// TwinCAT 3 PLC project MomTest
// Title: RIC_MOM
// Company: CFI
// Author: Phillip Prasinos
// ProjectVersion: 2.0.0
// Description: Mom Instance of RIC Gantry Crane
// ProgramVersion: 3.1.4020.2
// libraries:
//   Tc2_EtherCAT, * (Beckhoff Automation GmbH)
//   Tc2_MC2, * (Beckhoff Automation GmbH)
//   Tc2_SerialCom, * (Beckhoff Automation GmbH)
//   Tc2_Standard, * (Beckhoff Automation GmbH)
//   Tc2_System, * (Beckhoff Automation GmbH)
//   Tc2_SystemCX, * (Beckhoff Automation GmbH)
//   Tc2_Utilities, * (Beckhoff Automation GmbH)
//   Tc3_Interfaces, * (Beckhoff Automation GmbH)
//   Tc3_Module, * (Beckhoff Automation GmbH)
//   Tc2_System,3.4.17.0,Beckhoff Automation GmbH
// project tree:
//   DUTs/ EtherCAT_Kid.TcDUT, Patient.TcDUT
//   / FastTask.TcTTO, ParameterWriter.TcTTO
//   GVLs/ GVL_HMI.TcGVL
//   POUs/Function Blocks/ FB_CheckIn_EtherCAT.TcPOU, FB_EtherCATWriter.TcPOU, FB_HomeGantry.TcPOU, FB_Pulse.TcPOU, F_LoadDriveParameters.TcPOU, JoyStickGantryLogic.TcPOU, WirelessMove.TcPOU, P_FastTask.TcPOU
//   POUs/ HMIUpdate.TcPOU, MAIN.TcPOU, PlcTask.TcTTO, VariableValidation.TcPOU, WriteEtherCAT.TcPOU
//   POUs/Serial/ FB_SerialCom_Kiosk.TcPOU, FB_SerialCom_Remote.TcPOU, P_SerialRemote.TcPOU
// real-time tasks:
//   TASK PlcTask: cycle T#3ms, priority 2, ADS port 350
//   TASK ParameterWriter: cycle T#3ms, priority 6, ADS port 351
//   TASK FastTask: cycle T#4ms, priority 4, ADS port 352
// I/O:
//   DEVICE Device 3 (EtherCAT), AmsNetId 0.0.0.0.4.1
//     Box 1 (CX9020 EtherCAT slave) [CX9020 EtherCAT slave]
//     Box 2 (CX9020 EtherCAT slave) [CX9020 EtherCAT slave]
//     Box 3 (CX9020 EtherCAT slave) [CX9020 EtherCAT slave] (disabled)
//     Box 4 (CX9020 EtherCAT slave) [CX9020 EtherCAT slave] (disabled)
// variable links:
//   MomTest/MomTest Instance <-> Device 3 (EtherCAT)/Box 1 (CX9020 EtherCAT slave)
//     PlcTask Inputs/MAIN.JoyStickData <-> IO Inputs/Pdo Entry 11
//     PlcTask Inputs/MAIN.Kid[1].Address <-> IO Inputs/Pdo Entry 10
//     PlcTask Inputs/MAIN.Kid[1].HomedPosition_toMom <-> IO Inputs/Pdo Entry 2
//     PlcTask Inputs/MAIN.Kid[1].IsHardDownLimitReached <-> IO Inputs/Pdo Entry 5
//     PlcTask Inputs/MAIN.Kid[1].IsHardUpLimitReached <-> IO Inputs/Pdo Entry 4
//     PlcTask Inputs/MAIN.Kid[1].IsUltimateLimitReached <-> IO Inputs/Pdo Entry 3
//     PlcTask Inputs/MAIN.Kid[1].KidEstopCode <-> IO Inputs/Pdo Entry 9
//     PlcTask Inputs/MAIN.Kid[1].Load <-> IO Inputs/Pdo Entry 7
//     PlcTask Inputs/MAIN.Kid[1].MotionControllerErrorCode <-> IO Inputs/Pdo Entry 6
//     PlcTask Inputs/MAIN.Kid[1].Speed <-> IO Inputs/Pdo Entry 8
//     PlcTask Inputs/MAIN.Kid[1].UpdateWord_toMom <-> IO Inputs/Pdo Entry 1
//     PlcTask Outputs/MAIN.Kid[1].IsUltimateLimitBypassed <-> IO Outputs/Pdo Entry 6
//     PlcTask Outputs/MAIN.Kid[1].UpdateWord_FromMom <-> IO Outputs/Pdo Entry 1
//     PlcTask Outputs/MAIN.Kid[1].modeAccel_FromMom_Raw <-> IO Outputs/Pdo Entry 5
//     PlcTask Outputs/MAIN.Kid[1].modeDecel_FromMom_Raw <-> IO Outputs/Pdo Entry 7
//     PlcTask Outputs/MAIN.Kid[1].modeVel_FromMom_Raw <-> IO Outputs/Pdo Entry 4
//     PlcTask Outputs/MAIN.Kid[1].targetpos_FromMom_Raw <-> IO Outputs/Pdo Entry 2
//   MomTest/MomTest Instance <-> Device 3 (EtherCAT)/Box 2 (CX9020 EtherCAT slave)
//     PlcTask Inputs/MAIN.Kid[2].Address <-> IO Inputs/Pdo Entry 10
//     PlcTask Inputs/MAIN.Kid[2].HomedPosition_toMom <-> IO Inputs/Pdo Entry 2
//     PlcTask Inputs/MAIN.Kid[2].IsHardDownLimitReached <-> IO Inputs/Pdo Entry 5
//     PlcTask Inputs/MAIN.Kid[2].IsHardUpLimitReached <-> IO Inputs/Pdo Entry 4
//     PlcTask Inputs/MAIN.Kid[2].IsUltimateLimitReached <-> IO Inputs/Pdo Entry 3
//     PlcTask Inputs/MAIN.Kid[2].KidEstopCode <-> IO Inputs/Pdo Entry 9
//     PlcTask Inputs/MAIN.Kid[2].Load <-> IO Inputs/Pdo Entry 7
//     PlcTask Inputs/MAIN.Kid[2].MotionControllerErrorCode <-> IO Inputs/Pdo Entry 6
//     PlcTask Inputs/MAIN.Kid[2].Speed <-> IO Inputs/Pdo Entry 8
//     PlcTask Inputs/MAIN.Kid[2].UpdateWord_toMom <-> IO Inputs/Pdo Entry 1
//     PlcTask Outputs/MAIN.Kid[2].IsUltimateLimitBypassed <-> IO Outputs/Pdo Entry 6
//     PlcTask Outputs/MAIN.Kid[2].UpdateWord_FromMom <-> IO Outputs/Pdo Entry 1
//     PlcTask Outputs/MAIN.Kid[2].modeAccel_FromMom_Raw <-> IO Outputs/Pdo Entry 5
//     PlcTask Outputs/MAIN.Kid[2].modeDecel_FromMom_Raw <-> IO Outputs/Pdo Entry 7
//     PlcTask Outputs/MAIN.Kid[2].modeVel_FromMom_Raw <-> IO Outputs/Pdo Entry 4
//     PlcTask Outputs/MAIN.Kid[2].targetpos_FromMom_Raw <-> IO Outputs/Pdo Entry 2
//   MomTest/MomTest Instance <-> Device 3 (EtherCAT)/Box 3 (CX9020 EtherCAT slave)
//     PlcTask Inputs/MAIN.Kid[3].Address <-> IO Inputs/Pdo Entry 10
//     PlcTask Inputs/MAIN.Kid[3].HomedPosition_toMom <-> IO Inputs/Pdo Entry 2
//     PlcTask Inputs/MAIN.Kid[3].IsHardDownLimitReached <-> IO Inputs/Pdo Entry 5
//     PlcTask Inputs/MAIN.Kid[3].IsHardUpLimitReached <-> IO Inputs/Pdo Entry 4
//     PlcTask Inputs/MAIN.Kid[3].IsUltimateLimitReached <-> IO Inputs/Pdo Entry 3
//     PlcTask Inputs/MAIN.Kid[3].KidEstopCode <-> IO Inputs/Pdo Entry 9
//     PlcTask Inputs/MAIN.Kid[3].Load <-> IO Inputs/Pdo Entry 7
//     PlcTask Inputs/MAIN.Kid[3].MotionControllerErrorCode <-> IO Inputs/Pdo Entry 6
//     PlcTask Inputs/MAIN.Kid[3].Speed <-> IO Inputs/Pdo Entry 8
//     PlcTask Inputs/MAIN.Kid[3].UpdateWord_toMom <-> IO Inputs/Pdo Entry 1
//     PlcTask Outputs/MAIN.Kid[3].IsUltimateLimitBypassed <-> IO Outputs/Pdo Entry 6
//     PlcTask Outputs/MAIN.Kid[3].UpdateWord_FromMom <-> IO Outputs/Pdo Entry 1
//     PlcTask Outputs/MAIN.Kid[3].modeAccel_FromMom_Raw <-> IO Outputs/Pdo Entry 5
//     PlcTask Outputs/MAIN.Kid[3].modeDecel_FromMom_Raw <-> IO Outputs/Pdo Entry 7
//     PlcTask Outputs/MAIN.Kid[3].modeVel_FromMom_Raw <-> IO Outputs/Pdo Entry 4
//     PlcTask Outputs/MAIN.Kid[3].targetpos_FromMom_Raw <-> IO Outputs/Pdo Entry 2
//   MomTest/MomTest Instance <-> Device 3 (EtherCAT)/Box 4 (CX9020 EtherCAT slave)
//     PlcTask Inputs/MAIN.Kid[4].Address <-> IO Inputs/Pdo Entry 10
//     PlcTask Inputs/MAIN.Kid[4].HomedPosition_toMom <-> IO Inputs/Pdo Entry 2
//     PlcTask Inputs/MAIN.Kid[4].IsHardDownLimitReached <-> IO Inputs/Pdo Entry 5
//     PlcTask Inputs/MAIN.Kid[4].IsHardUpLimitReached <-> IO Inputs/Pdo Entry 4
//     PlcTask Inputs/MAIN.Kid[4].IsUltimateLimitReached <-> IO Inputs/Pdo Entry 3
//     PlcTask Inputs/MAIN.Kid[4].KidEstopCode <-> IO Inputs/Pdo Entry 9
//     PlcTask Inputs/MAIN.Kid[4].Load <-> IO Inputs/Pdo Entry 7
//     PlcTask Inputs/MAIN.Kid[4].MotionControllerErrorCode <-> IO Inputs/Pdo Entry 6
//     PlcTask Inputs/MAIN.Kid[4].Speed <-> IO Inputs/Pdo Entry 8
//     PlcTask Inputs/MAIN.Kid[4].UpdateWord_toMom <-> IO Inputs/Pdo Entry 1
//     PlcTask Outputs/MAIN.Kid[4].IsUltimateLimitBypassed <-> IO Outputs/Pdo Entry 6
//     PlcTask Outputs/MAIN.Kid[4].UpdateWord_FromMom <-> IO Outputs/Pdo Entry 1
//     PlcTask Outputs/MAIN.Kid[4].modeAccel_FromMom_Raw <-> IO Outputs/Pdo Entry 5
//     PlcTask Outputs/MAIN.Kid[4].modeDecel_FromMom_Raw <-> IO Outputs/Pdo Entry 7
//     PlcTask Outputs/MAIN.Kid[4].modeVel_FromMom_Raw <-> IO Outputs/Pdo Entry 4
//     PlcTask Outputs/MAIN.Kid[4].targetpos_FromMom_Raw <-> IO Outputs/Pdo Entry 2

CONFIGURATION MomTest
    RESOURCE PLC ON TwinCAT3
        TASK FastTask(INTERVAL := T#4ms, PRIORITY := 4);
        TASK ParameterWriter(INTERVAL := T#3ms, PRIORITY := 6);
        TASK PlcTask(INTERVAL := T#3ms, PRIORITY := 2);
        PROGRAM P_FastTask WITH FastTask : P_FastTask;
        PROGRAM WriteEtherCAT WITH ParameterWriter : WriteEtherCAT;
        PROGRAM MAIN WITH PlcTask : MAIN;
    END_RESOURCE
END_CONFIGURATION

// ---- DUTs/EtherCAT_Kid.TcDUT
TYPE EtherCAT_Kid :
STRUCT
	////////EtherCAT MoeAbsolute
	AxisID : INT := 0;
	//Status : FB_INIT_EtherCAT;
	//ReadStatus : FB_ReadStatus_EtherCAT := Status;
	//NcToPLC: FB_NcToPLC_Ethercat;
	
	//axisMoveAbs : FB_MoveAbsolute_EtherCAT;
	CheckIn : FB_CheckIn_EtherCAT;
	//ParameterReader : FB_EtherCATReader;
	//modeVel : DINT; //for hmi only

	// 1: System error sent from MOM
	
	//TargetPos : DINT;  //target position for move
	
	//modeAcc : DINT; //Maximum allowed Acceleration
	//modeJerk: UINT:= 80; //Maximum change in Accel per loop
	modeWindow : DINT:= 2000; //Allowed window for move to be complete
	leaveEnabled : BOOL := FALSE;
	//isBusy : BOOL := FALSE;
	//StartBit: BOOL :=FALSE;
	//RawToUU: LREAL;
//Velocity mode	profile EtherCAT Actual Values

	

	//VelDem_UU : DINT;
//Limits
	//dnUpLimit : DINT;
	//dnDownLimit: DINT;
	


	
	
	//HomeOffset_UU_R AT %I* : DINT;
	//HomeOffset_UU_W AT %Q* : DINT;
	

	CheckInt : DINT;
	bComTimeOutError : BOOL;
	//currentPosition: DINT;
	
	   RMT_EstopActivate : BOOL;
  RMT_DeadManPressed : BOOL;
  
  //EtherCAT 
    SetAdminMin : BOOL;
  SetAdminMax : BOOL;
  	  ResetCom : BOOL;
  SafteyReset : BOOL;
	UpdateWord_toMom  AT %I* : UDINT;
	HomedPosition_toMom AT %I* : DINT;
	IsUltimateLimitReached AT %I* : BYTE;
	IsHardUpLimitReached AT %I* : BYTE;
	IsHardDownLimitReached AT %I* : BYTE;
	MotionControllerErrorCode AT %I* :  UINT;


	 Load AT %I* : DINT;
	 Speed AT %I* :DINT;
	
	 KidEstopCode AT %I* : DINT;
	 		 Address AT %I*: AMSADDR;
	modeVel_FromMom : DINT;
modeAccel_FromMom : DINT;
ModeDecel_FromMom : DINT;
ScalingNumber : INT := 100; 		 
	 UpdateWord_FromMom AT %Q* : UDINT; //UpdateWord sends boolean information every cycle for quick inputs like deadman and Estop
	 targetpos_FromMom_Raw AT %Q* : DINT ; //FROM MOM
	 modeVel_FromMom_Raw AT %Q* : DINT ; //FROM MOM
	 modeAccel_FromMom_Raw AT %Q* : DINT ;
	 modeDecel_FromMom_Raw AT %Q* : DINT ;
	 IsUltimateLimitBypassed AT %Q* : BYTE;
	byPassSoftUp : BOOL;
	byPassSoftDown : BOOL;
	byPassHardup : BOOL;
	byPassHardDown : BOOL;
	byPassUltimate : BOOL;
	
	
	 //PAccel AT %I* : DINT  ;  //0x6048 vl_veloctity_acceleration
	// pDecel AT %I* : DINT ; //0x6049 vl_velocity_deceleration
	 //pVelMax AT %I* : INT; // 0x6042 vl_target_velocity
	 //OpModeCMD AT %I* : USINT := 2;; // 0x6060 Page 39 MODES OF OPERATION COMMAND 2-vl velocity mode  7 = interpolated position mode
 //pVelDem	AT %Q* : INT;
	// statusWord  AT %Q* : BITARR16; //0x6041
	// actualPos AT %Q*: DINT;// 0x6064 Position_actual_value
	// actualVel AT %Q*: DINT;
	// OpModeAct AT %Q* : USINT; // 0x6061 Page 39 MODES OF OPERATION DISPLAY read only result of changing 0x6060
	// ErrorCode AT %Q* : UINT;
	 
END_STRUCT
END_TYPE

// ---- DUTs/Patient.TcDUT
TYPE Patient :
STRUCT
	X : DINT := -10000; //patient location in mm
	Y : DINT := -10000; //patient location in mm
	ActiveSwitch: BOOL;
	AgeTimer : TON;
	AGE: TIME := T#0S;
END_STRUCT
END_TYPE

// ---- GVLs/GVL_HMI.TcGVL
{attribute 'qualified_only'}
VAR_GLOBAL PERSISTENT
	

//GantryLockWindow : DINT := 400;



//Patient{BeaconNumber}.Y
//Patient{BeaconNumber}.Active
//unJoystick1SelectNum : UINT;
//unJoystick2SelectNum : UINT;

//unJoystick1SelectNum : UINT;
//unJoystick2SelectNum : UINT;


//JoyStick1ScreenState : UINT;
//JoyStick2ScreenState : UINT;
//JoyStick1ScreenStateCommanded : INT;
//JoyStick2ScreenStateCOmmanded : INT;
//JoyStick1DeadManState : BOOL;
//JoyStick2DeadManState : BOOL;
//Joystick1ZAxisPressed : BOOL;
//JoyStick2ZAxisPressed : BOOL;
//JoyStick1SyncPressed : BOOL;
//JoyStick2SyncPressed: BOOL;
//JoyStick1Estop : BOOL;
//Joystick2Estop : BOOL;
//JoyStick1Age : TIME;
//JoyStick2Age : TIME;


//Bantry2BeaconNumber : INT;



GlobalFault_Code : INT;

GUIGlobalReset : BOOL;

	
END_VAR

VAR_GLOBAL
KioskScreenPower AT %Q* : BOOL;	
//Patient1 : Patient;
//Patient2 : Patient;
//Patient3 : Patient;
//Patient4 : Patient;
	EstopLight AT %Q* : BOOL;
Mom_Estop_Signal AT %I* : BOOL;
Kiosk_Estop_Signal AT %I* : BOOL;
END_VAR

// ---- POUs/Function Blocks/P_FastTask.TcPOU
PROGRAM P_FastTask
VAR
	
END_VAR

//MAIN.Serial1();
//MAIN.Serial2();
//MAIN.SerialRemoteFar(JoyStickNumber := GVL_HMI.unJoystick1SelectNum, Timeout := T#10S, ScreenActive => GVL_HMI.JoyStick1ScreenState);
//MAIN.SerialRemoteNear(JoyStickNumber := GVL_HMI.unJoystick2SelectNum, Timeout := T#10S, ScreenActive => GVL_HMI.JoyStick2ScreenState);

END_PROGRAM

// ---- POUs/WriteEtherCAT.TcPOU
PROGRAM WriteEtherCAT
VAR
	i : INT;
	i2 : INT;
	NetIDString : STRING;
	SymInfo  : ARRAY[1..4]  OF PLC_ReadSymInfoByName;
	SymInd : ARRAY[1..4] OF INT;
	HostFind : FB_GetHostAddrByName;
	COERead : adsread;
	Exec : BOOL;
	destaf : DINT;
END_VAR

//HostFind(sHostName := 'GANTRYKID_1', bExecute := Exec);
//FOR i := 1 TO 4 DO		
//	NetIDString :=INT_TO_STRING(BYTE_TO_INT(main.Kid[i].Address.netId[0]));
//
//	FOR i2 := 1 TO 5 DO NetIDString := CONCAT(Concat(netIDString, '.'), INT_TO_STRING(BYTE_TO_INT(main.Kid[i].Address.netId[i2]))); END_FOR
//SymInfo[i](NetID := NetIDString,  PORT:= main.kid[i].address.port, SymName:= 'TIID^Device 3 (EtherCAT Slave)^Outputs^CurrentPosition_ToMom', Start:=Exec);

	//MAIN.Kid[i].EtherCATWriter();
//END_FOR 	
//COERead(netid:=NetIDString, Port:=851, IDxGRP:=50593872,idxoffs:= 2164260877,Len:=4,DestAddr:=ADR(destaf),read:=Exec);

END_PROGRAM

// ---- POUs/MAIN.TcPOU
 PROGRAM MAIN
VAR_INPUT PERSISTENT
	Kid : ARRAY [1..6] OF EtherCAT_Kid;

END_VAR

VAR_INPUT
	JoyStickData AT %I* : DINT;
	JoyStickReading : DINT;
	ck : int;
	tcRestart : PLC_Reset;
		NumKids : INT := 2;
	GlobalEstopActive : BOOL;
	GlobalEstopCode : INT;
	GlobalEstopReason : STRING(255);
	JoyStickEstopActive : BOOL;
	StartHome1 : BOOL;
	Homing_Active : BOOL;
	StartHome2 : BOOL;
		xtar : DINT;
	ytar : DINT;
		JoyStick1DeadMan : BOOL;
	JoyStick2DeadMan : BOOL;
	jsResetter : BOOL;
	onUpLimit : BOOL;
	onDownLimit : BOOL;
END_VAR
VAR
	maxError : INT;
	ProcStart : NT_StartProcess;
	fbUpsPulse: FB_Pulse;

		MaxTimeOut_Reset : BOOL;
	fbWritePersistentData: FB_WritePersistentData;
		
	GantryCollision : BOOL;

	Mom_Estop_State : BOOL;
	//GantryClearanceWindow : DINT := 450;
	//HomeGantry : FB_HomeGantry;
	//HomeCarriage : FB_HomeGantry;
	TimeOutCheck : TIME;
	MaxTimeOut : Time;
	//	Kid : ARRAY [1..4] OF EtherCAT_Kid;
	//DeadMan : BOOL;
	//EStop : BOOL;
	//MAIN. : STRING(5000);
	
	i: DINT;
	Initialized : BOOL := FALSE;
	Serial1 : FB_SerialCom_Remote;
	Serial2 : FB_SerialCom_Kiosk;
	//Patient1 : Patient;
	//Patient2 : Patient;
	//Patient3 : Patient;
	//Patient4 : Patient;
	

	InterOpTimer : TON;
	TimeOutSwitch : BOOL;
	InterOpTimeout : BOOL;
	Execute : BOOL := true;
	GlobalReset : BOOL;
	ResetCount : INT;



	IN: INT;

	//HMIUpdate : HMIUpdate;
	//SerialRemoteFar : FB_SerialCom_Remote;
	//SerialRemoteNear : FB_SerialCom_Remote;
	
	//JS1 : JoyStickGantryLogic;
	//JS2 : JoystickGantryLogic;
	checker : DINT;
END_VAR



IF main.JoyStickEstopActive THEN main.GlobalEstopActive := TRUE;END_IF
IF NOT Initialized THEN
	//ProcStart(PathStr:='C:\users\administrator\desktop\setup.exe', dirname := 'C:\users\administrator\desktop', Start := TRUE);
	FOR i := 1 TO NumKids DO		
		MAIN.Kid[i].Checkin.KidID := DINT_TO_INT(i);	
		MAIN.Kid[i].AxisID := DINT_TO_INT(i); 
		KID[I].targetpos_FromMom_Raw := KID[I].HomedPosition_toMom;
		KID[i].leaveEnabled := FALSE;
	END_FOR 	
	Initialized := TRUE;
	RETURN;
END_IF


//HMIUpdate();

InterOpTimer(IN:= TimeOutSwitch, PT:= T#1000S, Q=> InterOpTimeout, ET=> TimeOutCheck);

if MaxTimeOut_Reset then MaxTimeOut := T#0s; MaxTimeOut_Reset := FALSE; END_IF
IF TimeOutCheck > MaxTimeOut THEN MaxTimeout := TimeOutCheck; END_IF

IF NOT TimeOutSwitch THEN TimeOutSwitch := NOT InterOpTimeout OR NOT TimeOutSwitch; END_IF
IF InterOpTimeOut THEN GlobalEstopActive := TRUE; GlobalEstopReason := 'INTEROPTIMEOUT'; END_IF


Joystick1Deadman := Joystick1Deadman AND NOT InterOpTimeout;




FOR i := 1 TO NumKids DO
	//MAIN.Kid[i].targetpos_FromMom_Raw := MAIN.Kid[1].HomedPosition_toMom;

	IF JoyStickData > 98304 AND JoyStickData <> 10000 THEN 
		
		MAIN.Kid[i].RMT_DeadManPressed := TRUE; 
	ELSIF JoyStickData <> 10000 THEN
		MAIN.Kid[i].RMT_DeadManPressed := FALSE;
	END_IF
	
	IF JoyStickData > 98304 THEN 
			
			JoyStickReading := (JoyStickData -98304 - 10000);
			MAIN.Kid[1].modeVel_FromMom_Raw := ABS((JoyStickReading * 1500)/10000);
			MAIN.Kid[1].modeAccel_FromMom_Raw := 3 * (((ABS(JoyStickReading) * 1200)/10000) +20);
			MAIN.Kid[1].modeDecel_FromMom_Raw := 3 * 1200;
			MAIN.Kid[1].targetpos_FromMom_Raw := MAIN.Kid[1].HomedPosition_toMom + JoyStickReading/20;	
	END_IF
		
	IF MAIN.Kid[i].modeAccel_FromMom_Raw < 10 THEN Kid[i].modeAccel_FromMom_Raw := 10; END_IF 
	//IF globalestopactive THEN kid[i].targetpos_FromMom_Raw := kid[i].HomedPosition_toMom; END_IF
	IF GVL_HMI.GUIGlobalReset THEN GlobalReset := TRUE; GVL_HMI.GUIGlobalReset := FALSE; END_IF
	IF GlobalReset THEN
		MAIN.Kid[i].resetCOM := TRUE;
		MAIN.Kid[i].SafteyReset := TRUE;
		MAIN.Kid[i].bComTimeOutError := FALSE;
		Kid[i].RMT_EstopActivate :=Mom_Estop_State;
		InterOpTimeOut := FALSE;
		timeoutSwitch := FALSE;
		GlobalEstopActive := false;
		GlobalEstopCode := 0;
		joystickEstopActive := False;
	END_IF
	
	IF Execute THEN
		MAIN.Kid[i].CheckIn.momControl := TRUE;
		IF(TimeOutCheck > T#500MS ) THEN   //this is the maximum allowed timeout when a deadman is pressed
			MAIN.Kid[i].RMT_DeadManPressed := FALSE;
		END_IF
	ELSE
		MAIN.Kid[i].CheckIn.momControl := FALSE;
		MAIN.Kid[i].RMT_DeadManPressed := FALSE;
	END_IF
	
		MAIN.Kid[i].CheckIn();
END_FOR 

IF GlobalReset AND NOT 
((Kid[1].CheckIn.momControl_FromKid AND(MAIN.Kid[1].Checkin.SafteyTripped  OR kid[1].checkin.CommError_FromKid)) OR 
 (Kid[2].CheckIn.momControl_FromKid AND (Kid[2].Checkin.SafteyTripped OR kid[2].checkin.CommError_FromKid)) OR
//(Kid[3].CheckIn.momControl_FromKid AND(Kid[3].Checkin.SafteyTripped OR kid[3].checkin.CommError_FromKid)) OR
//(Kid[4].CheckIn.momControl_FromKid AND(Kid[4].Checkin.SafteyTripped OR kid[4].checkin.CommError_FromKid)) OR
//(Kid[5].CheckIn.momControl_FromKid AND(Kid[5].Checkin.SafteyTripped OR kid[5].checkin.CommError_FromKid)) OR
//(Kid[6].CheckIn.momControl_FromKid AND(Kid[6].Checkin.SafteyTripped OR kid[6].checkin.CommError_FromKid)) OR
						GlobalEstopActive)  THEN
	GlobalReset:= FALSE;
	ResetCount := 0;
ELSIF GlobalReset THEN
	GlobalEstopActive := FALSE;
	ResetCount := ResetCount + 1;
	IF ResetCount > 300 THEN GlobalReset := FALSE; ResetCount := 0; END_IF
END_IF



//JS1(HookX := kid[1], HookY := Kid[2], sm := SerialRemoteFar); js1.Patient[1] := GVL_HMI.Patient1; js1.Patient[2] := GVL_HMI.Patient2; js1.Patient[3] := GVL_HMI.Patient3; js1.Patient[4] := GVL_HMI.Patient4;
//JS2(HookX := kid[3], HookY := Kid[4], sm := SerialRemoteNear); js2.Patient[1] := GVL_HMI.Patient1; js2.Patient[2] := GVL_HMI.Patient2; js2.Patient[3] := GVL_HMI.Patient3; js2.Patient[4] := GVL_HMI.Patient4;

checker := checker + 1;

i :=  Kid[1].HomedPosition_toMom; i := Kid[1].targetpos_FromMom_Raw; i := Kid[1].ScalingNumber; i := Kid[1].modeAccel_FromMom_RAW; i := Kid[1].modeVel_FromMom_RAW; i := Kid[1].ModeDecel_FromMom_RAW;
i :=  Kid[2].HomedPosition_toMom;  i := Kid[2].targetpos_FromMom_Raw;i := Kid[2].ScalingNumber; i := Kid[2].modeAccel_FromMom_RAW; i := Kid[2].modeVel_FromMom_RAW; i := Kid[2].ModeDecel_FromMom_RAW;
i :=  Kid[3].HomedPosition_toMom;  i := Kid[3].targetpos_FromMom_Raw;i := Kid[3].ScalingNumber; i := Kid[3].modeAccel_FromMom_RAW; i := Kid[2].modeVel_FromMom_RAW; i := Kid[3].ModeDecel_FromMom_RAW;
i :=  Kid[4].HomedPosition_toMom; i := Kid[4].targetpos_FromMom_Raw;  i := Kid[4].ScalingNumber; i := Kid[4].modeAccel_FromMom_RAW; i := Kid[2].modeVel_FromMom_RAW; i := Kid[3].ModeDecel_FromMom_RAW;




i := MAIN.Kid[1].UpdateWord_toMom;
i := MAIN.Kid[2].UpdateWord_toMom;
i := MAIN.Kid[3].UpdateWord_toMom;
i := MAIN.Kid[4].UpdateWord_toMom;
i := MAIN.Kid[5].UpdateWord_toMom;
i := MAIN.Kid[6].UpdateWord_toMom;


WriteEtherCAT();

fbUpsPulse(bEnable:= TRUE, tTimeOn:= T#100MS, tTimeOff:= T#30S, bPulse=> );


	in := in + 1;
	
	i := 2;
	ck :=DINT_TO_INT(Kid[1].targetpos_FromMom_Raw );
IF MAIN.Kid[1].targetpos_FromMom_Raw < 0 THEN  MAIN.Kid[1].targetpos_FromMom_Raw := 0; END_IF
IF MAIN.Kid[1].targetpos_FromMom_Raw > 12000 THEN  MAIN.Kid[1].targetpos_FromMom_Raw := 0; END_IF

	FOR i := 1 TO NumKids DO
		
		IF ABS(MAIN.Kid[i].HomedPosition_toMom - MAIN.Kid[1].HomedPosition_toMom) > maxError THEN maxError := DINT_TO_INT(ABS(MAIN.Kid[i].HomedPosition_toMom - MAIN.Kid[1].HomedPosition_toMom)); END_IF
		MAIN.Kid[i].targetpos_FromMom_Raw := MAIN.Kid[1].targetpos_FromMom_Raw;
		MAIN.Kid[i].modeVel_FromMom_Raw := MAIN.Kid[1].modeVel_FromMom_Raw + (ABS((MAIN.Kid[i].HomedPosition_toMom - MAIN.Kid[1].HomedPosition_toMom)) MOD 100);
		MAIN.Kid[i].modeAccel_FromMom_Raw := MAIN.Kid[1].modeAccel_FromMom_Raw + ABS((MAIN.Kid[i].HomedPosition_toMom - MAIN.Kid[1].HomedPosition_toMom)) MOD 50;
		MAIN.Kid[i].modeDecel_FromMom_Raw := MAIN.Kid[1].modeDecel_FromMom_Raw + ABS((MAIN.Kid[i].HomedPosition_toMom - MAIN.Kid[1].HomedPosition_toMom)) MOD 50;
		MAIN.Kid[i].ScalingNumber := MAIN.Kid[1].ScalingNumber;
		MAIN.Kid[i].RMT_DeadManPressed := MAIN.Kid[1].RMT_DeadManPressed;
		onDownLimit := FALSE;
		onUpLimit := FALSE;
		IF(MAIN.Kid[i].IsHardDownLimitReached> 0 AND MAIN.Kid[i].targetpos_FromMom_Raw <= MAIN.Kid[1].targetpos_FromMom_Raw) THEN onDownLimit := TRUE; END_IF
		IF(MAIN.Kid[i].IsHardUpLimitReached > 0 AND MAIN.Kid[i].targetpos_FromMom_Raw >= MAIN.Kid[1].targetpos_FromMom_Raw) THEN onUpLimit := TRUE; END_IF
	END_FOR
	
	
	FOR i := 1 TO NumKids DO
		IF(onUpLimit OR onDownLimit) THEN 
		   MAIN.Kid[i].RMT_DeadManPressed := FALSE;
 // MAIN.GlobalEstopActive := TRUE;
		END_IF
	END_FOR
	
	IF JoyStickData = 10000 AND NOT jsResetter  THEN jsResetter :=TRUE; GlobalEstopActive := TRUE; jsResetter := TRUE; END_IF
	IF jsResetter AND JoyStickData <> 10000 THEN GlobalReset := TRUE; jsResetter := FALSE; END_IF
	//IF TimeOutCheck > T#60S THEN
	//	tcRestart(RESET := TRUE);
	//END_IF

END_PROGRAM

// ---- POUs/Function Blocks/FB_Pulse.TcPOU
FUNCTION_BLOCK FB_Pulse
VAR_INPUT
	bEnable		: BOOL;		//When TRUE, bPulse will be on for tTimeOn and off for tTimeOff
	tTimeOn		: TIME;		//Time bPulse is On
	tTimeOff	: TIME;		//Time bPulse is Off
END_VAR
VAR_OUTPUT
	bPulse		: BOOL;
END_VAR
VAR
	fbTON		: TON;
	fbTOF		: TOF;
END_VAR

(*
//*****************************************************************Notes**********************************************************\\



  
  
//*****************************************************************Revs**********************************************************\\
   (          who            )(    Date    ) (   Rev     ) (								Disc						)
     Chris Mauban			 	2016.05.06		0.00.01		Initial Code
				
     		 								 				
	 						
	
//*****************************************************************Code**********************************************************\\
*)
fbTON(IN:= bEnable AND NOT fbTOF.Q, PT:= tTimeOn, Q=> , ET=> );
fbTOF(IN:= fbTON.Q, PT:= tTimeOff, Q=> , ET=> );

IF bEnable THEN
	bPulse := fbTON.M;
ELSE
	bPulse := FALSE;
END_IF

END_FUNCTION_BLOCK

// ---- POUs/Serial/FB_SerialCom_Remote.TcPOU
FUNCTION_BLOCK FB_SerialCom_Remote

VAR
	x : INT :=0; 
	FRAME : ARRAY [1..10 ] OF BYTE ; 
	TxBuffer	: ComBuffer;
	RxBuffer	: ComBuffer;
		NextOffset : INT;
	yRead : INT;
	xRead : INT; 
	ButtonStateRead : INT;
	ScreenStateRead : INT;
	bCount: INT;
		(* background communication with the EL6001 terminal *)
	fbEL6002Ctrl		: SerialLineControl;
	(* 	I/O variables for a EL6001 terminal*)
	stIn_EL6002B AT %I*	: EL6inData22B;	(* linked to the EL6001 in the TwinCAT System Manager *)
	stOut_EL6002B AT %Q*	: EL6outData22B;(* linked to the EL6001 in the TwinCAT System Manager *)
	SendTimer		: TON;
	fbSend		: SendString;
	bSendBusy	: BOOL;
	eSendErrorID: ComError_t;
	fbReceive		: ReceiveData;
	AgeTimer : TON;
	Disconnected : BOOL;
	CalmDown : TIME := T#900MS;
END_VAR

VAR_INPUT
	Timeout : TIME := T#3S; //Timespan to concider the remote disconnected
	sSendString: STRING;
	ScreenCommanded : BYTE;
	JoyStickNumber : INT;
END_VAR

VAR_OUTPUT
	yAxis : INT:=0; //Up/Down result of Joystick 50 to -50
	xAxis : INT:=0; //Left/Right Result of Joystick 50 to -50
	DeadmanPressed: INT:=0; //Resulting consecutive frames with DeadmanPressed (Positive) or not pressed 
	EstopPressed: INT:=0; //Resulting consecutive frames with DeadmanPressed (Positive) or not pressed 
	ZAxisPressed: INT:=0; //Resulting consecutive frames with DeadmanPressed (Positive) or not pressed 
	SyncPressed : INT:=0; //Resulting consecutive frames with DeadmanPressed (Positive) or not pressed 
	Age : TIME;
	Connected : BOOL;
	ScreenActive : INT;
END_VAR


(* background communication with the EL6001 terminal *)
AgeTimer(IN:=TRUE, PT := Timeout, ET=> AGE, Q=> Disconnected); Connected := NOT Disconnected;

fbEL6002Ctrl(	Mode:= SERIALLINEMODE_EL6_22B, 	pComIn:= ADR(stIn_EL6002B),	pComOut:= ADR(stOut_EL6002B), 	SizeComIn:= SIZEOF(stIn_EL6002B), 	TxBuffer:= TxBuffer, 	RxBuffer:= RxBuffer, );

// Call the send block every second to repeat the transmission.
// Also call the block as long as it is busy to finish a transmission.
IF ScreenActive = ScreenCommanded OR LEN(sSendString)> 2 OR txbuffer.count > 5 THEN
	SendTimer(IN:=TRUE, PT := T#50MS + CalmDown);
	
	ELSE
	SendTimer(IN:=TRUE, PT := T#50MS );

END_IF
IF TXBuffer.Count > 10 THEN sSendString := ''; END_IF
IF SendTimer.Q OR bSendBusy THEN
	SendTimer(IN:=FALSE); (* reset timer *)
	fbSend(	SendString:=  sSendString,	TXbuffer:= TxBuffer,	Busy=> bSendBusy,	Error=> );
	IF fbSend.Error <> COMERROR_NOERROR THEN
		eSendErrorID := fbSend.Error;
	END_IF
END_IF


IF RxBuffer.Count > 9 THEN
	//IF LEN(sSendString) <= 1 THEN sSendString := ''; END_IF
	fbReceive(pReceiveData :=ADR(FRAME), SizeReceiveData := SIZEOF(FRAME),	 DataReceived =>,	 RxBuffer := RXBUFFER);
	FOR X := 1 TO 5 DO
		IF FRAME[x]= 116 AND FRAME[x+1] = 100 AND FRAME[x + 2]= 114 AND FRAME[x+3]=58  THEN sSendString := CONCAT(DINT_TO_STRING(100000 + JoyStickNumber), '$R$N');  END_IF //filter:
		IF FRAME[x]= 76 AND FRAME[x+1] = 79 AND FRAME[x + 2]= 83 AND FRAME[x+3]=83 THEN sSendString := CONCAT(DINT_TO_STRING(100000 + JoyStickNumber), '$R$N');  END_IF  //RF LOSS
		IF FRAME[x] = 10 AND FRAME[x+5] = 13 THEN
			//IF ScreenCommanded = 74 THEN sSendString := 'J' ; END_IF
sSendString := F_ToChR(ScreenCommanded); 
			
			yRead := FRAME[x+1] ;
			xRead := FRAME[x+2];
			ButtonStateRead := BYTE_TO_INT(Frame[x+3]);
			ScreenStateRead := Frame[x+4];
			
		//IF ((ButtonStateRead + xAxis + yAxis + ScreenStateRead) MOD 2)  = BOOL_TO_INT(ButtonStateRead > 64) THEN 
				ButtonStateRead := ButtonStateRead MOD 64;   //buttonstates 7th bit is used for parity 0==odd 1==even (64 = EVEN) 
				yAxis := yRead -150;
				xAxis := xRead - 150;
				NextOffSet := X;
				ScreenActive := ScreenStateRead;
				IF ButtonStateRead >= 32 THEN SyncPressed := BOOL_TO_INT(SyncPressed <=0) * (SyncPressed -1); ButtonStateRead := ButtonStateRead - 32; ELSE SyncPressed := BOOL_TO_INT(SyncPressed >=0) * (SyncPressed + 1); END_IF
				IF ButtonStateRead >= 16  THEN ZAxisPressed := BOOL_TO_INT(ZAxisPressed <=0) * (ZAxisPressed -1); ButtonStateRead := ButtonStateRead - 16; ELSE ZAxisPressed := BOOL_TO_INT(ZAxisPressed >=0) *(ZaxisPressed + 1); END_IF
				IF ButtonStateRead < 8  THEN EstopPressed := BOOL_TO_INT(EstopPressed<= 0) * (EstopPressed -1);  ELSE EStopPressed := BOOL_TO_INT(EStopPressed >= 0) * (EStopPressed + 1); ButtonStateRead := (ButtonStateRead - 8); END_IF
				IF ButtonStateRead >= 3  THEN DeadManPressed :=  BOOL_TO_INT(DeadManPressed <= 0) *(DeadManPressed - 1); ButtonStateRead := ButtonStateRead - 4; ELSE DeadmanPressed := BOOL_TO_INT(DeadManPressed >= 0) * (DeadmanPressed + 1); END_IF
				IF SyncPressed > 100 THEN SyncPressed := 100; END_IF; IF SyncPressed < -100 THEN SyncPressed := -100; END_IF
				IF ZAxisPressed > 1000 THEN ZAxisPressed := 100; END_IF; IF ZAxisPressed < -1000 THEN ZAxisPressed := -100; END_IF
				IF EStopPressed > 1000 THEN EStopPressed := 100; END_IF; IF EStopPressed < -1000 THEN EStopPressed := -100; END_IF
				IF DeadManPressed > 1000 THEN DeadManPressed := 100; END_IF; IF DeadManPressed < -1000 THEN DeadManPressed := -100; END_IF
				AgeTimer(in:=False);
			//FRAME[X+ 1] :=0; FRAME[X+ 2] :=0; FRAME[X+ 3] :=0; FRAME[X+ 4] :=0; FRAME[X+ 5] :=0;
		//	ELSE 
					bCount := bCount +1;
					
					
			//END_IF
			
			
		END_IF
		FRAME[X] :=0;
	END_FOR

END_IF

IF AgeTimer.Q THEN 
	ScreenActive := 72;
	//ScreenCommanded := 72; 
	sSendString := CONCAT(DINT_TO_STRING(100000 + JoyStickNumber), '$R$N');
ELSIF sCREENcOMMANDED = 72 THEN
	//ScreenCommanded := 73;
 END_IF
//	Age := Age + T#1MS; //IF THIS IS NOT THE CYCLE TIME OF THE TASK IT WILL NOT BE ACCURATE;

IF ScreenActive = 0 THEN ScreenActive := 72; END_IF

END_FUNCTION_BLOCK

// ---- POUs/Serial/FB_SerialCom_Kiosk.TcPOU
FUNCTION_BLOCK FB_SerialCom_Kiosk

VAR
	begpack : bool;
	x : INT;
	prefix : STRING := '$R$N';
	suffix : STRING := '$R$N';
	fcount : DINT :=0;
	FRAME : ARRAY [1..200 ] OF BYTE ; 
	swCheck0 : STRING;
	swCheck1 : STRING;
	swCheck2 : STRING;
	swCheck3 : STRING;
	swCheck4 : STRING;
	swCheck5 : STRING;
	ReceiveByte : ReceiveByte;
	LastReceivedByte : BYTE;
	TxBuffer	: ComBuffer;
	RxBuffer	: ComBuffer;

		(* background communication with the EL6001 terminal *)

		fbEL6002Ctrl		: SerialLineControl;
	bEL6002CtrlError	: BOOL;
	eEL6002CtrlErrorID	: ComError_t;
	(* 	I/O variables for a EL6001 terminal*)
	stIn_EL6002 AT %I*	: EL6inData22B;	(* linked to the EL6001 in the TwinCAT System Manager *)
	stOut_EL6002 AT %Q*	: EL6outData22B;(* linked to the EL6001 in the TwinCAT System Manager *)
	stIn_EL6002B AT %I*	: EL6inData22B;	(* linked to the EL6001 in the TwinCAT System Manager *)
	stOut_EL6002B AT %Q*	: EL6outData22B;(* linked to the EL6001 in the TwinCAT System Manager *)
	Timer		: TON;
	fbSend		: SendString;
	bSendBusy	: BOOL;
	eSendErrorID: ComError_t;

	fbReceive		: ReceiveData;
fbReceivestr		: ReceiveSTRING;


	eReceiveErrorID	: ComError_t;
	nReceiveCounter	: UDINT;

	fbF_Trig: F_TRIG;
	nStringLength: INT;
	sStringWithoutPrefix: STRING(255);

END_VAR

VAR_INPUT
	bEnable : BOOL;
	sSendString: STRING;
END_VAR

VAR_OUTPUT
	bStringReceived	: BOOL;
	sReceivedString	: STRING;
	sLastReceivedString: STRING := 'NULL';
	bDone : BOOL;
END_VAR

(*
The SerialLineControl function block is supposed to be called in every PLC cycle.
It communicates with the serial line hardware device and transmits or receives data.
The SerialLineControl can be called in the standard task (e.g.for PcCOM port usage) 
or in a separate fast task (e.g.for terminal usage) as well.
A fast separate task will be necessary at high baud rates or with KL6001 terminals 
which have a small process image (3 or 5 data bytes only)
*)

(* background communication with the EL6001 terminal *)

fbEL6002Ctrl(
	Mode:= SERIALLINEMODE_EL6_22B, 
	pComIn:= ADR(stIn_EL6002), 
	pComOut:= ADR(stOut_EL6002), 
	SizeComIn:= SIZEOF(stIn_EL6002), 
	Error=> , 
	ErrorID=> , 
	TxBuffer:= TxBuffer, 
	RxBuffer:= RxBuffer, );
IF fbEL6002Ctrl.Error THEN
	bEL6002CtrlError := TRUE;
	eEL6002CtrlErrorID := fbEL6002Ctrl.ErrorID;
END_IF


// Call the send block every second to repeat the transmission.
// Also call the block as long as it is busy to finish a transmission.
Timer(IN:=bEnable, PT := T#125MS);
IF Timer.Q OR bSendBusy THEN
	Timer(IN:=FALSE); (* reset timer *)
	fbSend(	SendString:= sSendString,
			TXbuffer:= TxBuffer,
			Busy=> bSendBusy,
			Error=> );
	IF fbSend.Error <> COMERROR_NOERROR THEN
		eSendErrorID := fbSend.Error;
	END_IF
END_IF

fbF_Trig(CLK:=bSendBusy);
bDone := bSendBusy;
	
//	Receive string data:
//	The block receives any data strings beginning with a STX ($02) and ending with an ETX ($03) character.	
//fbEL6002Ctrl.RxBuffer.Count

WHILE RxBuffer.Count > 205 AND ReceiveByte.ReceivedByte <> 150  DO			
	ReceiveByte( RxBuffer := RXBuffer);
END_WHILE

IF RxBuffer.Count > 199 THEN
fbReceive(//pPrefix := ADR(prefix),
		  //psuffix := ADR(SUFFIX),
		 //LenPrefix := 2,
		 pReceiveData :=ADR(FRAME),
		 SizeReceiveData := SIZEOF(FRAME),
		 DataReceived =>,
		 RxBuffer := RXBUFFER);
		 END_IF
		 
	IF (Frame[1] = 78 OR frame[2] = 78 OR frame[3] = 78) AND NOT GVL_HMI.KioskScreenPower  THEN
		GVL_HMI.KioskScreenPower := TRUE;
	ELSIF (Frame[1] = 70 OR frame[2] = 70 OR frame[3] = 70) AND  GVL_HMI.KioskScreenPower  THEN
			GVL_HMI.KioskScreenPower := FALSE;

	END_IF



(*
fbReceivestr(
	Prefix:= '$N',//'$02',
	Suffix:= '$R',//'$03',
	Timeout:= T#1s,
	ReceivedString:= sReceivedString,
	RXbuffer:= RxBuffer,
	StringReceived=> bStringReceived,
	Busy=> bReceiveBusy,
	Error=> ,
	RxTimeout=> bReceiveTimeout );





	//ReceiveByte(RxBuffer := RXBuffer);
	
		begPack := FALSE;
	 //CLEAR OUT BUFFER TO PREVENT OVERRUN
		ReceiveByte( RxBuffer := RXBuffer);
		IF ReceiveByte.ReceivedByte = 13 THEN
			swCheck2 := BYTE_TO_STRING(ReceiveByte.ReceivedByte);
			WHILE RxBuffer.Count > 5 AND begpack = FALSE DO //CLEAR OUT BUFFER TO PREVENT OVERRUN
				
					begPack := TRUE;
					fcount := fcount + 1;
					
					ELSE
					
							swCheck1 := BYTE_TO_STRING(ReceiveByte.ReceivedByte);
					fcount := fcount - 1;
				END_IF
			END_WHILE
			ELSE
				swCheck3 := BYTE_TO_STRING(ReceiveByte.ReceivedByte);

		END_IF
	END_WHILE
	

	
	IF begPack AND RxBuffer.Count > 4 THEN
		
				ReceiveByte( RxBuffer := RXBuffer);
				//swCheck2 := BYTE_TO_STRING(ReceiveByte.ReceivedByte);
				IF ReceiveByte.ByteReceived  AND ReceiveByte.ReceivedByte > 50 THEN yRead := BYTE_TO_INT(ReceiveByte.ReceivedByte) ; END_IF
				ReceiveByte(RxBuffer := RXBuffer);
				//swCheck3 := BYTE_TO_STRING(ReceiveByte.ReceivedByte);
				IF ReceiveByte.ByteReceived  AND ReceiveByte.ReceivedByte >50 THEN xRead := BYTE_TO_INT(ReceiveByte.ReceivedByte) ; END_IF
				ReceiveByte( RxBuffer := RXBuffer);
				//swCheck4 := BYTE_TO_STRING(ReceiveByte.ReceivedByte);
				IF ReceiveByte.ByteReceived AND ReceiveByte.ReceivedByte <>0 THEN ButtonStateRead := BYTE_TO_INT(ReceiveByte.ReceivedByte); END_IF
				ReceiveByte( RxBuffer := RXBuffer);
				//swCheck5 := BYTE_TO_STRING(ReceiveByte.ReceivedByte);
				IF ReceiveByte.ByteReceived  AND ReceiveByte.ReceivedByte <>0 THEN ScreenStateRead :=BYTE_TO_INT(ReceiveByte.ReceivedByte); END_IF
	END_IF
	

*)


	


IF fbReceivestr.Error <> COMERROR_NOERROR THEN
	eReceiveErrorID := fbReceivestr.Error;
END_IF

IF bStringReceived THEN
	nReceiveCounter := nReceiveCounter + 1;
	sStringWithoutPrefix := sReceivedString;
	nStringLength := LEN(sStringWithoutPrefix);
	sLastReceivedString := sStringWithoutPrefix;	
END_IF

END_FUNCTION_BLOCK

// ---- POUs/Function Blocks/FB_CheckIn_EtherCAT.TcPOU
FUNCTION_BLOCK FB_CheckIn_EtherCAT

VAR_INPUT
	GlobalGo : BOOL;
	momControl: BOOL;
momControl_FromKid: BOOL;
	KidID : INT := -1;
	//UpdateWord_toKid AT %Q* : UDINT;
	//UpdateWord_FromKid AT %I* : UDINT;
	SafteyTripped : BOOL; //DEADMAN STATE OF MOM
	Hard_Limit_Tripped : BOOL;
		HomeOperation_Active : BOOL;
END_VAR

VAR_OUTPUT
	Kid_EstopPressed : BOOL;
	CommError_FromKid : BOOL;
		CollisionSwitch : BOOL; 
		HomeActivated : BOOL;
END_VAR

VAR
	UltimateByPassCounter : INT;
	checkid : UINT;
	checkingInt : UDINT := 0;
	SysTime : GetSystemTime();
	Unknown: BOOL;
	LeaveEnabled: BOOL;
	heartBeat : BOOL;
	KidComTimer : TON;
	KidCom_ET : TIME;
		SoftLimitCounter : INT;
	
	RMT_EstopActivate : BOOL;
	Ultimate_Tripped : BOOL;	

	//SafteyTripped: INT;
END_VAR



IF MAIN.Kid[KidID].modeAccel_FromMom_Raw = 0 THEN MAIN.Kid[KidID].modeAccel_FromMom_Raw := 10; END_IF
checkingInt := MAIN.Kid[KidID].UpdateWord_ToMom;
 		 
		checkingInt := checkingInt MOD 1024;
		Kid_EstopPressed := CheckingInt/512 > 0; CheckingInt := CheckingInt MOD 512;
	Ultimate_Tripped := CheckingInt/256 > 0; CheckingInt := CheckingInt MOD 256;
	momControl_FromKid:= checkingInt / 128 > 0;	checkingInt := checkingInt MOD 128;
	CollisionSwitch := checkingInt / 64 > 0;	
	checkingInt := checkingInt MOD 64;
	HomeActivated := checkingInt / 32 > 0;			checkingInt := checkingInt MOD 32;
	CommError_FromKid:= checkingInt / 16 > 0;	checkingInt := checkingInt MOD 16;
	SafteyTripped := checkingInt / 8 > 0;	checkingInt := checkingInt MOD 8;
	Hard_Limit_Tripped:= checkingInt / 4 > 0;	checkingInt := checkingInt MOD 4;
	LeaveEnabled:= FALSE;
	KidComTimer(IN:=checkingInt MOD 2 >0 = HeartBeat OR MAIN.GlobalReset, PT:=T#150MS , Q=> CommError_FromKid, ET=> KidCom_ET );
	HeartBeat :=checkingInt MOD 2>0;
	
	IF NOT momcontrol_Fromkid THEN RETURN; END_IF
	
	IF KidID = -1 THEN RETURN; END_IF
	IF NOT MomControl THEN RETURN; END_IF
IF SafteyTripped THEN 
	MAIN.GlobalEstopActive :=  NOT MAIN.Kid[KidID].SafteyReset; 
	
	IF MAIN.GlobalEstopCode = 0 THEN 
		MAIN.GlobalEstopCode :=  LREAL_TO_INT(EXPT(2, KidID-1)); 
		IF CommError_FromKid OR MAIN.Kid[KidID].bComTimeOutError  THEN MAIN.GlobalEstopCode := MAIN.GlobalEstopCode + 16; END_IF;
		IF Ultimate_Tripped THEN Main.GlobalEstopCode := Main.GlobalEstopCode + 32; END_IF;
		IF MAIN.InterOpTimeout THEN MAIN.GlobalEstopCode := Main.GlobalEstopCode + 64; END_IF
		//IF SafteyTripped THEN MAIN.GlobalEstopCode := main.GlobalEstopCode + 128; END_IF
		IF NOT GVL_HMI.Mom_Estop_Signal OR NOT GVL_HMI.Kiosk_Estop_Signal THEN MAIN.GlobalEstopCode := Main.GlobalEstopCode + 256; END_IF
		IF main.JoyStickEstopActive THEN main.GlobalEstopCode := main.GlobalEstopCode + 512; END_IF
	END_IF
	
END_IF

	IF CommError_FromKid THEN
		MAIN.GlobalEstopActive := NOT MAIN.Kid[KidID].SafteyReset;
	END_IF
	

	IF MAIN.Kid[KidID].resetCOM  THEN
		CommError_FromKid := FALSE;
	END_IF
	

	RMT_Estopactivate := (Main.GlobalEstopActive AND NOT MAIN.Kid[KidID].SafteyReset) OR NOT GVL_HMI.Mom_Estop_Signal OR NOT GVL_HMI.Kiosk_Estop_Signal;
	unknown := FALSE;
	//LeaveEnabled := TRUE;
	MAIN.Kid[KidID].UpdateWord_FromMom:=	(INT_TO_UDINT(KidID) * 134217728) +
	(BOOL_TO_UDINT(MAIN.Kid[KidID].byPassSoftDown) * 16384) +
	(BOOL_TO_UDINT(MAIN.Kid[KidID].byPassSoftUp) * 8192) +
	(BOOL_TO_UDINT(MAIN.Kid[KidID].byPassHardDown) * 4096) +
	(BOOL_TO_UDINT(MAIN.Kid[KidID].byPassHardup) * 2048) +
	(BOOL_TO_UDINT(MAIN.Kid[KidID].byPassUltimate) * 1024 ) +
						(BOOL_TO_UDINT(HomeOperation_Active) * 512) +
						(BOOL_TO_UDINT(MAIN.GantryCollision) * 256) +
						(BOOL_TO_UDINT(momControl) * 128) +
						(BOOL_TO_UDINT(MAIN.Kid[KidID].RMT_DeadManPressed OR main.Kid[kidid].CheckIn.HomeOperation_Active) * 64) +
						(BOOL_TO_UDINT(MAIN.Kid[KidID].SafteyReset) * 32) +
						(BOOL_TO_UDINT(MAIN.Kid[KidID].resetCOM) * 16) +
						(BOOL_TO_UDINT(MAIN.GlobalEstopActive AND NOT MAIN.GlobalReset) * 8) +
						(BOOL_TO_UDINT(FALSE) * 4) +
						(BOOL_TO_UDINT(LeaveEnabled) * 2) +
						BOOL_TO_UDINT(HeartBeat);
	
	//IF MAIN.Kid[KidID].SetAdminMin OR MAIN.Kid[KidID].SetAdminMax THEN
	//	SoftLimitCounter := SoftLimitCounter + 1;
	//	IF SoftLimitCounter > 1000 THEN MAIN.Kid[KidID].SetAdminMax := FALSE; MAIN.Kid[KidID].SetAdminMin := FALSE; 	MAIN.kid[kidid].IsUltimateLimitBypassed := FALSE; END_IF	
	//END_IF
	
MAIN.Kid[KidID].SafteyReset := MAIN.Kid[KidID].SafteyReset AND SafteyTripped;
MAIN.Kid[KidID].resetCOM := MAIN.Kid[KidID].resetCOM AND ( MAIN.Kid[KidID].bComTimeOutError OR CommError_FromKid);

		MAIN.Kid[KidID].bComTimeOutError := CommError_FromKid;
		Main.GlobalEstopActive := momcontrol_fromkid AND (Main.GlobalEstopActive OR  SafteyTripped);
		
//IF MAIN.kid[Kidid].IsUltimateLimitBypassed THEN 
//	UltimateByPassCounter := UltimateByPassCounter + 1;
//	IF 	UltimateByPassCounter > 100000 THEN MAIN.kid[Kidid].isultimatelimitbypassed := FALSE; UltimateByPassCounter :=0; END_IF
		
//	END_IF
//MAIN.Kid[KidID].SafteyReset := Estop_Activate;
									
						
//	MAIN.Kid[KidID].modeVel_FromMom_Raw := (MAIN.Kid[KidID].modeVel_FromMom ;
//IF KidId = 3 THEN MAIN.Kid[KidID].modeVel_FromMom_Raw := (MAIN.Kid[KidID].modeVel_FromMom  * main.Kid[KidID].ScalingNumber)/115; END_IF
//MAIN.Kid[KidID].modeAccel_FromMom_Raw := (MAIN.Kid[KidID].modeAccel_FromMom/2) + (MAIN.Kid[KidID].modeAccel_FromMom  * main.Kid[KidID].ScalingNumber/200)	;
//IF KidId = 3 THEN MAIN.Kid[KidID].modeAccel_FromMom_Raw := (MAIN.Kid[KidID].modeAccel_FromMom/2) + (MAIN.Kid[KidID].modeAccel_FromMom  * main.Kid[KidID].ScalingNumber/205)	; END_IF
//;
//MAIN.Kid[KidID].modeDecel_FromMom_Raw :=  MAIN.Kid[KidID].modeDEcel_FromMom;

(*IF MAIN.Kid[KidID].modeVel_FromMom_Raw > 0 THEN
	IF Main.Kid[kidID].HomedPosition_toMom < 5 THEN MAIN.Kid[KidID].modeVel_FromMom_Raw := 2; END_IF
ELSE
	IF Main.Kid[kidID].HomedPosition_toMom < 100 THEN MAIN.Kid[KidID].modeVel_FromMom_Raw := -5 *(MAIN.Kid[KidID].modeVel_FromMom_Raw/10); END_IF
END_IF*)

END_FUNCTION_BLOCK

// ---- POUs/Function Blocks/FB_EtherCATWriter.TcPOU
FUNCTION_BLOCK FB_EtherCATWriter
VAR_INPUT
	KidID : INT :=0;
	IDToWrite : USINT :=0;
	lrEncoder_ScalingNum : LREAL;
	Admin_Min :DINT;
	Admin_Max :DINT;
	Direction_Flipped : BOOL;
	lrDistance_1_Motor_Rev : LREAL;
	QuickStop_Accel : DINT;
	lrDecel_For_EStop : DINT;
	ParameterID_ToKid AT %Q* : USINT := 1;
	ParameterID_FromKid AT %I* : USINT;
	
END_VAR
VAR_OUTPUT
//	WrittenAll : BOOL := FALSE;
END_VAR

VAR
	

	DataInt : DINT;
	RecievedData : ARRAY [1..256] OF INT; //used to count reads of each parameter
	
	
END_VAR

IF KidID = 0 THEN RETURN; END_IF
//ParameterWord_FromMom consists of 32 bytes. The first(greatest) 8 bytes ID the Variable to write and the last 24 include the data. 
// ParameterID		Parameter To Write					Format
// 1				GVL_Motion.lrEncoder_ScalingNum		1/DATAINT := ScalingNum
// 2				GVL_Index.Admin_Max					:= 512 * DataInt (largest bit is sign)	
// 3				GVL_Index.Admin_Min					:= 	512 * DataInt (largest bit is sign)	
// 4				GVL_Index.Direction_Flipped			>0 		
// 5				GVL_Motion.lrDistance_1_Motor_Rev	:= ?????????????????????????
// 6				GVL_Speeds.QuickStop_Accel		
// 7 				GVL_Speeds.lrDecel_For_EStop		:=?
 ParameterID_ToKid := IDToWrite;

CASE IDToWrite OF
//1: 	MAIN.Kid[KidID].ParameterWord_ToKid := LREAL_TO_DINT(lrEncoder_ScalingNum) ;
//2: 	MAIN.Kid[KidID].ParameterWord_ToKid := Admin_Max ;
//3: 	MAIN.Kid[KidID].ParameterWord_ToKid := Admin_Min ;
//4:  MAIN.Kid[KidID].ParameterWord_ToKid := BOOL_TO_INT(Direction_Flipped) ;
//5: 	MAIN.Kid[KidID].ParameterWord_ToKid := LREAL_TO_DINT(lrDistance_1_Motor_Rev) ;
//6:	MAIN.Kid[KidID].ParameterWord_ToKid := QuickStop_Accel ;
//7:	MAIN.Kid[KidID].ParameterWord_ToKid := lrDecel_For_EStop ;
//8:  MAIN.Kid[KidID].ParameterWord_ToKid  := MAIN.Kid[KidID].maxVelRef;
ELSE
	IDToWrite := 0;
END_CASE

IF ParameterID_FromKid = ParameterID_ToKid THEN
	IDToWrite := IDToWrite + 1;
	ELSIF IDToWrite = 0 THEN
		//IDToWrite := 1;
END_IF

//IF MAIN.Kid[KidID].ParameterWord_ToKid < 16777216 THEN
//	MAIN.Kid[KidID].ParameterWord_ToKid  := MAIN.Kid[KidID].ParameterWord_ToKid + (16777216 * IDToWrite);
//END_IF
//RecievedData[ID] := RecievedData[ID] + 1;

END_FUNCTION_BLOCK

// ---- POUs/Function Blocks/FB_HomeGantry.TcPOU
FUNCTION_BLOCK FB_HomeGantry
VAR_INPUT
	Enable : BOOL;
	KidID : INT;
	HomeStart : BOOL;
	OffHome : BOOL;
	KidStart : DINT;
	CaseNum : DINT;
	PrevVel : DINT; 
END_VAR
VAR_OUTPUT
END_VAR
VAR

END_VAR

IF  KidID = 0 THEN RETURN; END_IF

IF NOT enable OR MAIN.GlobalEstopActive THEN
	main.Kid[kidid].TargetPos := main.Kid[kidID].currentPosition;
END_IF

IF HomeStart THEN
	PrevVel := MAIN.Kid[KidID].modeVel;
	KidStart := MAIN.Kid[KidID].currentPosition;
	MAIN.Kid[KidID].CheckIn.HomeOperation_Active := TRUE;
	HomeStart := FALSE;
	OffHome := FALSE;
	CaseNum := 0;
END_IF


CASE CaseNum OF
	0:
		IF KidID = 1 THEN MAIN.Kid[KidID].TargetPos := KidStart + 100; END_IF
		IF KidID = 3 THEN MAIN.Kid[KidID].TargetPos := KidStart - 100; END_IF
		IF KidID = 2 THEN MAIN.Kid[KidID].TargetPos := KidStart + 100; END_IF
		IF KidID = 4 THEN MAIN.Kid[KidID].TargetPos := KidStart + 100; END_IF
		
		MAIN.Kid[KidID].modeVel := MAIN.Kid[KidID].HomeSpeed;
		IF MAIN.Kid[KidID].CheckIn.HomeActivated  THEN 
			CaseNum := CaseNum + 1; 
		ELSIF ABS(MAIN.Kid[KidID].currentPosition - MAIN.Kid[KidID].TargetPos) < 10 THEN 
			CaseNum := CaseNum + 2; 
		END_IF
	1: 
		IF KidID = 1 THEN MAIN.Kid[KidID].TargetPos := MAIN.Kid[KidID].currentPosition + 100; END_IF
		IF KidID = 3 THEN MAIN.Kid[KidID].TargetPos := MAIN.Kid[KidID].currentPosition - 100; END_IF
		IF KidID = 2 THEN MAIN.Kid[KidID].TargetPos := KidStart + 1000; END_IF
		IF KidID = 4 THEN MAIN.Kid[KidID].TargetPos := KidStart + 1000; END_IF
		
		IF (KidID = 1 OR KidId = 3) AND NOT MAIN.Kid[KidID].CheckIn.HomeActivated OR MAIN.GantryCollision  THEN CaseNum := CaseNum + 1; END_IF
		IF (KidID = 2 OR KidId = 4) AND MAIN.Kid[KidID].CheckIn.Hard_Limit_Tripped  THEN  CaseNum := CaseNum + 1; END_IF
	2: 
		IF KidID = 3 THEN MAIN.Kid[KidID].TargetPos := MAIN.Kid[KidID].currentPosition + 100; END_IF
		IF KidID = 1 THEN MAIN.Kid[KidID].TargetPos := MAIN.Kid[KidID].currentPosition - 100; END_IF
		
		IF (KidID = 1 OR KidID = 3) AND MAIN.Kid[KidID].CheckIn.HomeActivated  THEN 
			MAIN.Kid[KidID].modeVel := MAIN.Kid[KidID].HomeSpeed/3;
			CaseNum := CaseNum + 1;
		ELSIF (KidID = 2 OR KidID = 4) AND MAIN.Kid[KidID].CheckIn.Hard_Limit_Tripped THEN
			MAIN.Kid[KidID].CheckIn.HomeOperation_Active := FALSE;
			CaseNum := CaseNum + 2;
		END_IF
			
	3: 
		IF KidID = 3 THEN MAIN.Kid[KidID].TargetPos := MAIN.Kid[KidID].currentPosition + 100; END_IF
		IF KidID = 1 THEN MAIN.Kid[KidID].TargetPos := MAIN.Kid[KidID].currentPosition - 100; END_IF
		IF NOT MAIN.Kid[KidID].CheckIn.HomeActivated  THEN 
			MAIN.Kid[KidID].CheckIn.HomeOperation_Active := FALSE;
			CaseNum := CaseNum + 1;
		END_IF
	4: 	
		//IF KidID = 1 THEN MAIN.Kid[KidID].TargetPos := 0; END_IF;
	   //	IF KidID = 3 THEN MAIN.Kid[KidID].TargetPos := 3295; END_IF;
		//IF  ABS(MAIN.Kid[KidID].currentPosition - MAIN.Kid[KidID].TargetPos) < 10 THEN
			MAIN.Kid[KidID].TargetPos := MAIN.Kid[KidID].currentPosition;
			Enable := FALSE;
				Main.Kid[kidid].modeVel := DINT_TO_UINT(prevVel);
			KidID := 0;
			
		
		//	MAIN.Kid[KidID].RMT_DeadManPressed := FALSE;
		//	CaseNum := CaseNum + 1;
		//END_IF
	5: 
	
END_CASE

END_FUNCTION_BLOCK

// ---- POUs/Function Blocks/F_LoadDriveParameters.TcPOU
FUNCTION F_LoadDriveParameters : BOOL //Places the correct values into MOMs placeholder variables for transmission to each kid;
VAR_INPUT
	KidID : INT; //Axis identifier for each kid for which we will load parameters
	AxisID : INT;
END_VAR
VAR
END_VAR

	(*

CASE AxisID OF
	1:
	MAIN.Kid[KidID].EtherCATWriter.lrEncoder_ScalingNum := 3020;
	MAIN.Kid[KidID].EtherCATWriter.Admin_Min :=1000;
	MAIN.Kid[KidID].EtherCATWriter.Admin_Max :=100000;
	MAIN.Kid[KidID].EtherCATWriter.Direction_Flipped := 0;
	MAIN.Kid[KidID].EtherCATWriter.lrDistance_1_Motor_Rev :=300;
	MAIN.Kid[KidID].EtherCATWriter.QuickStop_Accel := 6000;
	MAIN.Kid[KidID].EtherCATWriter.lrDecel_For_EStop := 9000;
	
	2:
	MAIN.Kid[KidID].EtherCATWriter.lrEncoder_ScalingNum := 2000;
	MAIN.Kid[KidID].EtherCATWriter.Admin_Min :=1000;
	MAIN.Kid[KidID].EtherCATWriter.Admin_Max :=100000;
	MAIN.Kid[KidID].EtherCATWriter.Direction_Flipped := 0;
	MAIN.Kid[KidID].EtherCATWriter.lrDistance_1_Motor_Rev :=300;
	MAIN.Kid[KidID].EtherCATWriter.QuickStop_Accel := 6000;
	MAIN.Kid[KidID].EtherCATWriter.lrDecel_For_EStop := 9000;
	
END_CASE*)

END_FUNCTION

// ---- POUs/Function Blocks/JoyStickGantryLogic.TcPOU
FUNCTION_BLOCK JoyStickGantryLogic
VAR_INPUT
	HookX : EtherCAT_Kid;
	HookY : EtherCAT_Kid;
	MaxTime : TIME;
	Patient : ARRAY[0..4] OF patient;
	ModeCheck : DINT;
END_VAR

VAR_IN_OUT
		sm : FB_SerialCom_Remote; //SerialRemote Assigned to Gantry
END_VAR

VAR_OUTPUT
	TrackedPatient : INT;
END_VAR

VAR
WirelessMove : WirelessMove;
X: INT;
DeadManState : BOOL;

END_VAR
////Patient1 : Patient;
//Patient2 : Patient;
//Patient3 : Patient;
//Patient4 : Patient;

IF sm.SyncPressed = 5  THEN
	GVL_HMI.GUIGlobalReset := TRUE;
	RETURN;
END_IF


IF MAIN.GlobalEstopActive THEN
	sm.ScreenCommanded := 51; 
	TrackedPatient := 0;
	RETURN;
ELSE
	IF sm.ScreenCommanded = 51 THEN sm.ScreenCommanded := 73; END_IF
END_IF


IF sm.ScreenActive =73 OR sm.ScreenActive = 74 OR sm.ScreenActive = 72 THEN
	

	sm.ScreenCommanded := 73;
	FOR X := 1 TO 4 DO
		IF ((Patient[x].X - HookX.currentPosition) * (Patient[x].X - HookX.currentPosition)) + ((Patient[x].Y - HookY.currentPosition) * (Patient[x].Y - HookY.currentPosition)) >0 THEN
			IF SQRT(((Patient[x].X - HookX.currentPosition) * (Patient[x].X - HookX.currentPosition)) + ((Patient[x].Y - HookY.currentPosition) * (Patient[x].Y - HookY.currentPosition))) < GVL_HMI.GantryLockWindow 
				AND Patient[x].AGE < T#500MS THEN
				sm.ScreenCommanded := 74;
				IF sm.ZAxisPressed > 1 AND sm.DeadmanPressed < 0 AND sm.ScreenActive = 74 THEN
					TrackedPatient := X;
					sm.ScreenCommanded := 74+ INT_TO_BYTE(X);
				END_IF
			END_IF
		END_IF
	END_FOR

END_IF

IF sm.ZAxisPressed > 2 AND sm.DeadmanPressed > 2 THEN TrackedPatient := 0; sm.ScreenCommanded := 74; END_IF

IF sm.DeadmanPressed >= 2 AND sm.ScreenActive < 75 AND sm.ScreenCommanded > 71 THEN
	ModeCheck := 1;
	WirelessMove(HookX := HookX, HookY:= HookY, sm :=SM, WindowScaling := 1);
	DeadmanState := TRUE;
ELSIF sm.DeadmanPressed < 1 AND sm.ScreenActive > 74 AND sm.ScreenCommanded > 74  AND patient[TrackedPatient].AGE < T#500MS AND sm.Age < T#1000MS THEN
		ModeCheck := 2;
	DeadmanState := TRUE;
	MAIN.Kid[Hookx.CheckIn.KidID].TargetPos := Patient[TrackedPatient].X;
	MAIN.Kid[HookY.CheckIn.KidID].TargetPos := Patient[TrackedPatient].Y;
ELSIF sm.DeadmanPressed < 0 THEN
		ModeCheck := 3;
	DeadManState := FALSE;
ELSE
		ModeCHeck := 4;

END_IF


x:= TrackedPatient;
IF TrackedPatient <> 0 THEN
	IF( Patient[x].x < -500 OR Patient[x].x > 3900 OR Patient[x].y > 9500 OR Patient[x].y < -500 OR sm.Age > T#2000MS OR Patient[x].AGE > T#500MS) THEN
		ModeCheck := ModeCheck + 10;
		sm.ScreenCommanded := 73;
		TrackedPatient := 0;
	END_IF
	if patient[x].Age > MaxTime then Maxtime := Patient[x].AGE; END_IF
END_IF



IF sm.EstopPressed > 1 THEN
	MAIN.JoyStickEstopActive := TRUE;
	
END_IF


IF HookX.CheckIn.KidID = 1 THEN
	MAIN.JoyStick1DeadMan:=DeadmanState;
ELSE
	MAIN.JoyStick2DeadMan := DeadmanState;
END_IF

END_FUNCTION_BLOCK

// ---- POUs/Function Blocks/WirelessMove.TcPOU
FUNCTION_BLOCK WirelessMove 
VAR_INPUT

	sm : FB_SerialCom_Remote; //SerialRemote Assigned to Gantry
	WindowScaling : INT := 1; //Scaling Factor for target window distance
END_VAR
VAR
	XTar : DINT;
	YTar : DINT;
END_VAR
VAR_IN_OUT
		HookX : EtherCat_Kid;
	HookY : EtherCat_Kid;
END_VAR

IF sm.DeadmanPressed >=1 AND SM.Age < T#800MS THEN
	IF Hookx.currentPosition + (((ABS(sm.xAxis) * sm.xAxis) * WindowScaling) / -50) > -1000000 OR Hookx.currentPosition + (((ABS(sm.xAxis) * sm.xAxis) * WindowScaling) / -50) < 1000000 THEN
		XTar := Hookx.currentPosition + (((ABS(sm.xAxis) * sm.xAxis) * WindowScaling) / -50);
	END_IF
	IF HookY.currentPosition + (((ABS(sm.YAxis) * sm.YAxis) * WindowScaling) / -25) > -1000000 OR HookY.currentPosition + (((ABS(sm.YAxis) * sm.YAxis) * WindowScaling) / -25) < 100000 THEN
			YTar := HookY.currentPosition + (((ABS(sm.YAxis) * sm.YAxis) * WindowScaling) / -25);
	END_IF

	main.XTAR := xtar;
	main.YTar := Ytar;
	Main.Kid[hookX.CheckIn.KidID].TargetPos := XTar;
	Main.Kid[Hooky.CheckIn.KidID].TargetPos := YTar;
	//HookY.TargetPos := YTar;
	ELSE
		Main.Kid[hookX.CheckIn.KidID].TargetPos := Main.Kid[hookX.CheckIn.KidID].Currentposition;
		Main.Kid[Hooky.CheckIn.KidID].TargetPos := Main.Kid[Hooky.CheckIn.KidID].CurrentPosition;

END_IF

END_FUNCTION_BLOCK

// ---- POUs/HMIUpdate.TcPOU
FUNCTION_BLOCK HMIUpdate
VAR_INPUT
	
END_VAR
VAR_OUTPUT
END_VAR
VAR
	i : INT;
	LoopCounter : INT;
	UltimateByPassCounter : INT;
	
	
	
	Active: INT;
END_VAR



GVL_HMI.GlobalFault_Code := MAIN.GlobalEstopCode;

IF MAIN.GlobalEstopActive THEN
	LoopCounter := LoopCounter + 1;
	ELSE
	loopcounter := 0;
END_IF

IF LoopCounter = 0 OR LoopCounter > 400 THEN
	GVL_HMI.EstopLight := TRUE;
END_IF

IF LoopCounter > 800 THEN
	LoopCounter := 0;
	GVL_HMI.EstopLight := FALSE;
END_IF

GVL_HMI.Patient1.AgeTimer(IN:= NOT GVL_HMI.Patient1.ActiveSwitch, PT:= T#5S, ET=>GVL_HMI.Patient1.AGE);
GVL_HMI.Patient2.AgeTimer(IN:= NOT GVL_HMI.Patient2.ActiveSwitch, PT:= T#5S, ET=>GVL_HMI.Patient2.AGE);
GVL_HMI.Patient3.AgeTimer(IN:= NOT GVL_HMI.Patient3.ActiveSwitch, PT:= T#5S, ET=>GVL_HMI.Patient3.AGE);
GVL_HMI.Patient4.AgeTimer(IN:= NOT GVL_HMI.Patient4.ActiveSwitch, PT:= T#5S, ET=>GVL_HMI.Patient4.AGE);
 GVL_HMI.Patient1.ActiveSwitch := FALSE;
 GVL_HMI.Patient2.ActiveSwitch:= FALSE;
//IF NOT GVL_HMI.Patient2.ActiveSwitch THEN GVL_HMI.Patient2.ActiveSwitch := TRUE; END_IF
//IF NOT GVL_HMI.Patient3.ActiveSwitch THEN GVL_HMI.Patient3.ActiveSwitch:= TRUE; END_IF
GVL_HMI.Patient3.ActiveSwitch:= FALSE;
GVL_HMI.Patient4.ActiveSwitch:= FALSE;
//IF NOT GVL_HMI.Patient4.ActiveSwitch THEN GVL_HMI.Patient4.ActiveSwitch:= TRUE; END_IF


GVL_HMI.JoyStick1ScreenStateCommanded := main.SerialRemoteNear.ScreenCommanded;
GVL_HMI.JoyStick2ScreenStateCOmmanded := MAIN.SerialRemoteFar.ScreenCommanded;
GVL_HMI.JoyStick1DeadManState := main.SerialRemoteNear.DeadmanPressed>0;
GVL_HMI.JoyStick2DeadManState := MAIN.SerialRemoteFar.DeadmanPressed>0;
GVL_HMI.Joystick1ZAxisPressed := MAIN.SerialRemoteNear.ZAxisPressed>0;
GVL_HMI.JoyStick2ZAxisPressed :=MAIN.SerialRemoteFar.ZAxisPressed>0;
GVL_HMI.JoyStick1SyncPressed := MAIN.SerialRemoteNear.SyncPressed>0;
GVL_HMI.JoyStick2SyncPressed:= MAIN.SerialRemoteFar.SyncPressed>0;
GVL_HMI.JoyStick1Estop := main.SerialRemoteNear.EstopPressed>0;
GVL_HMI.Joystick2Estop := MAIN.SerialRemoteFar.EstopPressed>0;
GVL_HMI.JoyStick1Age := MAIN.SerialRemoteNear.Age;
GVL_HMI.JoyStick2Age := MAIN.SerialRemoteFar.Age;

END_FUNCTION_BLOCK

// ---- POUs/Serial/P_SerialRemote.TcPOU
(*
SerialCom_InfoSys_Sample1 (v2.0)
This sample sends and receives a string via serial communication.
Hardware interface used: EL terminal
*)
PROGRAM P_SerialRemote
VAR
	fbEL600x	: FB_SerialCom;
	sMyString: STRING;
	

	sMyStringSend: STRING  := '1';

	bStartTimer: BOOL;
	nLEDSend: INT;
	btest: BOOL;
	fbTOF: TOF;
	fbTON: Ton;
	fbTONZon: Ton;
	fbTONHeartbeatON: Ton;
	fbTONHeartbeatOFF: Ton;
	bLastCount: BOOL;
	unStringSize: UINT;
	sStringDecipher : STRING;
	fbTOFDevOn: TOF;
	i: INT;
	sSerialStringList: ARRAY[1..20] OF STRING;
	fbTonSerialStream: TON;
	bJoystickTimeoutReset: BOOL;
	fbTONSend: TON;
	sTempSendString: STRING;
	fbR_Trig: R_TRIG;
	fbTONResend: TON;
	sScreenDrawTemp: STRING;
	arrStringDraw: ARRAY[1..20] OF STRING;
	arrStringDrawCnt: INT;
	nScreenDrawnMult: INT;
END_VAR

fbTOFDevOn(IN:= fbEL600x.bStringReceived, PT:= T#1S);
GVL_Serial.bDeviceOn := INT_TO_BOOL(STRING_TO_INT(F_ToCHR(sMyString[1]))) AND fbTOFDevOn.Q;

//////////////////////////////////////////////////////
//Disable all Wireless Inputs when GVL_PLC.bLocalKeySwitchInput is FALSE
//////////////////////////////////////////////////////
IF GVL_PLC.bLocalKeySwitchInput THEN
	sMyString := fbEL600x.sLastReceivedString;
ELSE
	sMyString := '';
END_IF
//////////////////////////////////////////////////////

unStringSize := SIZEOF(sMyString);

IF P_JoystickSetup.bTurnOffJoystickSend OR GVL_PLC.bWiredJoystickEn THEN
	sMyStringSend := P_JoystickSetup.sSendString;
	GVL_Serial.bEstop := FALSE;
	GVL_Serial.bDeviceOn := FALSE;
ELSE
	IF fbEL600x.nStringLength = 36 AND unStringSize = 81 THEN
	//V10502v H10508h ZFz DFd EFe CFc J0002j
		//Vertical Signal
		IF F_ToCHR(sMyString[0]) = 'V' AND F_ToCHR(sMyString[6]) = 'v' THEN
			sStringDecipher := LEFT(sMyString,6);
			sStringDecipher := RIGHT(sStringDecipher,4);
			GVL_Serial.nVertical := STRING_TO_INT(sStringDecipher);
		END_IF
		
		//Horizontal Signal
		IF F_ToCHR(sMyString[7]) = 'H' AND F_ToCHR(sMyString[13]) = 'h' THEN
			sStringDecipher := LEFT(sMyString,13);
			sStringDecipher := RIGHT(sStringDecipher,4);
			GVL_Serial.nHorizontal := STRING_TO_INT(sStringDecipher);
		END_IF
		
		//Zon Signal
		IF F_ToCHR(sMyString[14]) = 'Z' AND F_ToCHR(sMyString[16]) = 'z' THEN
			sStringDecipher := LEFT(sMyString,16);
			sStringDecipher := RIGHT(sStringDecipher,1);
			GVL_Serial.bZonRaw := sStringDecipher = 'N';
		END_IF
		fbTONZon(IN:=GVL_Serial.bZonRaw,PT:=T#100MS);
		GVL_Serial.bZon := fbTONZon.Q;
		
		//Deadman Signal
		IF F_ToCHR(sMyString[17]) = 'D' AND F_ToCHR(sMyString[19]) = 'd' THEN
			sStringDecipher := LEFT(sMyString,19);
			sStringDecipher := RIGHT(sStringDecipher,1);
			GVL_Serial.bDeadmanRaw := sStringDecipher = 'N';
		END_IF
		fbTON(IN:=GVL_Serial.bDeadmanRaw,PT:=T#200MS);
		GVL_Serial.bDeadman := fbTON.Q;
		
		//Estop Signal
		IF F_ToCHR(sMyString[20]) = 'E' AND F_ToCHR(sMyString[22]) = 'e' THEN
			sStringDecipher := LEFT(sMyString,22);
			sStringDecipher := RIGHT(sStringDecipher,1);
			GVL_Serial.bEstop := sStringDecipher = 'F';
		END_IF
		//fbTOF(IN:=INT_TO_BOOL(STRING_TO_INT(MID(sMyString,1,23))),PT:=T#500MS);
		//GVL_Serial.bEstop := fbTOF.Q;
		
		//Heartbeat Count Signal
		IF F_ToCHR(sMyString[23]) = 'C' AND F_ToCHR(sMyString[25]) = 'c' THEN
			sStringDecipher := LEFT(sMyString,25);
			sStringDecipher := RIGHT(sStringDecipher,1);
			GVL_Serial.bCount := sStringDecipher = 'N';
		END_IF
		

		//Joystick Number
		IF F_ToCHR(sMyString[26]) = 'J' AND F_ToCHR(sMyString[31]) = 'j' THEN
			sStringDecipher := LEFT(sMyString,31);
			sStringDecipher := RIGHT(sStringDecipher,4);
			GVL_HMI.unJoystickCurrentNum := STRING_TO_UINT(sStringDecipher);
		END_IF
		
				//Joystick Screen Last Drawn
		IF F_ToCHR(sMyString[32]) = 'S' AND F_ToCHR(sMyString[34]) = 's' THEN
			sStringDecipher := LEFT(sMyString,34);
			sStringDecipher := RIGHT(sStringDecipher,1);
			GVL_Serial.sScreenDrawn := sStringDecipher;
			FOR nScreenDrawnMult := 2 TO 4 DO
				GVL_Serial.sScreenDrawn := CONCAT(GVL_Serial.sScreenDrawn, sStringDecipher);
			END_FOR
		END_IF
		
		//////////////////////////////////////////////////////////
		//OLED Screen
		/////////////////////////////////////////////////////////
		sMyStringSend := GVL_Serial.sJoystickScreen;
(*	IF GVL_Serial.bDeadmanRaw THEN
		sMyStringSend := 'FFFF';
	ELSE
		sMyStringSend := 'EEEE';
	END_IF
*)
		IF sMyStringSend <> sTempSendString THEN
			GVL_Serial.bSendJoystickModeEn := TRUE;
		END_IF
	END_IF
END_IF


//////////////////////////////////////////////////////////
//Serial Send Logic
/////////////////////////////////////////////////////////
fbTONSend(IN:= GVL_Serial.bSendJoystickModeEn, PT:= T#275MS);
//Send Last OLED Status change for 350MS before sending Sensor and Deadman Update
IF fbTONSend.Q THEN
	GVL_Serial.bSendJoystickModeEn := FALSE;
	sTempSendString := sMyStringSend;
END_IF

fbTONResend(IN:= GVL_Serial.bDeviceOn AND NOT GVL_Serial.bSendJoystickModeEn, PT:= T#500MS);
IF fbTONResend.Q THEN
	GVL_Serial.bSendJoystickModeEn := TRUE;
END_IF

fbEL600x(
//	bEnable := GVL_Serial.bDeviceOn OR P_JoystickSetup.bSendEn OR btest,
//	bEnable := P_JoystickSetup.bSendEn OR btest,
	bEnable := (GVL_Serial.bSendJoystickModeEn OR P_JoystickSetup.bSendEn OR btest) AND GVL_PLC.bLocalKeySwitchInput,
	sSendString := sMyStringSend,
	TxBuffer:= GVL_Serial.TxBufferEL,
	RxBuffer:= GVL_Serial.RxBufferEL);



//////////////////////////////////////////////////////////
//Serial Receive List
/////////////////////////////////////////////////////////	
IF fbEL600x.bStringReceived THEN
	FOR i:=1 TO 19 DO
		sSerialStringList[21-i] := sSerialStringList[20-i];
	END_FOR
	sSerialStringList[1] := fbEL600x.sReceivedString;
END_IF




//////////////////////////////////////////////////////////
//Serial Connection Timeout
/////////////////////////////////////////////////////////
//fbTonSerialStream(IN:= NOT fbEL600x.bStringReceived); //AND NOT fbTonSerialStream.Q, PT := T#5S);
fbTonSerialStream(IN:= NOT fbEL600x.bStringReceived AND NOT fbTonSerialStream.Q, PT := T#2S);
IF fbTonSerialStream.Q AND NOT (sSerialStringList[1] = 'TIMEOUT') THEN
	FOR i:=1 TO 19 DO
		sSerialStringList[21-i] := sSerialStringList[20-i];
	END_FOR
	sSerialStringList[1] := 'TIMEOUT';	
END_IF

//bJoystickTimeoutReset := GVL_PLC.unLastJoystick <> GVL_HMI.unJoystickCurrentNum;

fbTONHeartbeatON(IN:= GVL_Serial.bCount AND NOT bJoystickTimeoutReset, PT:= T#2000MS);
fbTONHeartbeatOFF(IN:= NOT GVL_Serial.bCount AND NOT bJoystickTimeoutReset, PT:= T#2000MS);
IF fbTONHeartbeatON.Q OR fbTONHeartbeatOFF.Q THEN
	GVL_Serial.bCommLoss := TRUE;
	GVL_Serial.bEstop := FALSE;
END_IF

//IF bJoystickTimeoutReset or
IF GVL_HMI.bGlobalReset THEN
	GVL_Serial.bCommLoss := FALSE;
END_IF

IF GVL_Serial.sScreenDrawn <> sScreenDrawTemp THEN
	FOR arrStringDrawCnt:=1 TO 19 DO
		arrStringDraw[21-arrStringDrawCnt] := arrStringDraw[20-arrStringDrawCnt];
	END_FOR
	arrStringDraw[1] := GVL_Serial.sScreenDrawn;
	sScreenDrawTemp := GVL_Serial.sScreenDrawn;	
END_IF

END_PROGRAM

// ---- POUs/VariableValidation.TcPOU
FUNCTION_BLOCK VariableValidation  //this code is only used to prevent TwinCAT's IDE from identifying variables as unused

VAR_INPUT
END_VAR
VAR_OUTPUT
END_VAR
VAR
END_VAR

GVL_HMI.JoyStick1ScreenStateCommanded := GVL_HMI.JoyStick1ScreenStateCommanded;
GVL_HMI.JoyStick2ScreenStateCOmmanded := GVL_HMI.JoyStick2ScreenStateCOmmanded;
GVL_HMI.JoyStick1DeadManState := GVL_HMI.JoyStick1DeadManState;
GVL_HMI.JoyStick2DeadManState :=GVL_HMI.JoyStick2DeadManState;
GVL_HMI.Joystick1ZAxisPressed := GVL_HMI.Joystick1ZAxisPressed;
GVL_HMI.JoyStick2ZAxisPressed := GVL_HMI.JoyStick2ZAxisPressed;
GVL_HMI.JoyStick1SyncPressed := GVL_HMI.JoyStick1SyncPressed ;
GVL_HMI.JoyStick2SyncPressed:= GVL_HMI.JoyStick2SyncPressed;
GVL_HMI.JoyStick1Estop := GVL_HMI.JoyStick1Estop;
GVL_HMI.Joystick2Estop := GVL_HMI.Joystick2Estop;
GVL_HMI.JoyStick1Age := GVL_HMI.JoyStick1Age;
GVL_HMI.JoyStick2Age := GVL_HMI.JoyStick2Age ;


//Bantry2BeaconNumber : INT;



GVL_HMI.GlobalFault_Code := GVL_HMI.GlobalFault_Code;

END_FUNCTION_BLOCK
